(* CODESYS project tc3_physics.library
   TcLibraryId: Beckhoff Automation GmbH|Tc3_Physics|3.1.10.3
   Company: Beckhoff Automation GmbH
   DefaultNamespace: Tc3_Physics
   Version: 3.1.10.3
   Placeholder: Tc3_Physics
   Title: Tc3_Physics

Project tree, tasks and I/O mapping:
  Version/
    global variables Global_Version
  POUs/
    _Internal/
      function block IPlcGeometry2D [ST]: FB_init, FB_exit
      function block IPlcDynamicConstraint [ST]: FB_init, FB_exit
    Spatial/
      Positions/
        function block PositionXY [ST]: FB_init, FB_reinit, FB_exit, SetZero, SetValues, SetValuesXY, SetValuesRP, GetRadius, GetPhi, Invert, ConcatenateWith, ShiftByXY, x, y
        function block PositionXYC [ST]: FB_init, FB_reinit, FB_exit, SetZero, SetValues, SetValuesXY, SetValuesXYC, Invert, ConcatenateWith, StepByLocalXY, ShiftByXY, TurnByC, Transform, x, y, c
    Dynamics/
      function block DynamicConstraint_Container [ST]: FB_init, FB_exit, Clear, AddConstraint, Count
      function block DynamicConstraint_PathXY [ST]: FB_init, FB_exit, SetValuesVADJ, V, A, D, J
      function block DynamicConstraint_Path [ST]: FB_init, FB_exit
      function block DynamicConstraint_Coordinates [ST]: FB_init, FB_exit, AddLimit, SetLimit, RemoveLimit, Clear, GetV, GetA, GetD, GetJ, Count
    Coordinates/
      function GetMcsCoordinateType [ST]
  DUTs/
    Enumerations/
      data type E_RotationCoordinates
      data type E_CoordCategory
      data type E_McsCoordType
    data type CoordinateType
  GVLs/
    global variables GVL
*)

// DUTs/CoordinateType

(* Coordinate type. Use provided constants such as Coord_Mcs_X or factory functions such as GetMcsCoordinateType for creation. *)
	{attribute 'TcIecLibraryType'}
{attribute 'Namespace' := 'MC'}
TYPE CoordinateType : 
	STRUCT
		(* Reserved. *)
		{attribute 'hide'}
		_reserved0 : ULINT := 0;
	END_STRUCT
END_TYPE

// DUTs/Enumerations/E_RotationCoordinates

(* Enumeration of rotation conventions. 
          The order of letters defines the order of rotation around local axes.
          This also defines order in which user should program rotation values. *)
	{attribute 'TcIecLibraryType'}
{attribute 'qualified_only'}
{attribute 'strict'}
TYPE E_RotationCoordinates : (
	ABC:=0, 	(* ABC *)
	ACB:=1, 	(* ACB *)
	BCA:=2, 	(* BCA *)
	BAC:=3, 	(* BAC *)
	CAB:=4, 	(* CAB *)
	CBA:=5, 	(* CBA *)
	ABA:=6, 	(* ABA *)
	ACA:=7, 	(* ACA *)
	BAB:=8, 	(* BAB *)
	BCB:=9, 	(* BCB *)
	CAC:=10, 	(* CAC *)
	CBC:=11	(* CBC *)
) UDINT;
END_TYPE

// DUTs/Enumerations/E_CoordCategory

(* Enumeration coordinate categories. *)
	{attribute 'TcIecLibraryType'}
{attribute 'qualified_only'}
{attribute 'strict'}
TYPE E_CoordCategory : (
	Invalid:=16#0, 	(* Invalid *)
	MCS:=16#1, 	(* MCS *)
	ACS:=16#2, 	(* ACS *)
	Uninterpreted:=16#3	(* Uninterpreted *)
) UDINT;
END_TYPE

// DUTs/Enumerations/E_McsCoordType

(* Enumeration of MCS coordinate types. *)
	{attribute 'TcIecLibraryType'}
{attribute 'qualified_only'}
{attribute 'strict'}
TYPE E_McsCoordType : (
	Invalid:=16#0, 	(* Invalid *)
	X:=16#11, 	(* X *)
	Y:=16#21, 	(* Y *)
	Z:=16#31, 	(* Z *)
	A1:=16#41, 	(* A1 *)
	A2:=16#42, 	(* A2 *)
	A3:=16#43, 	(* A3 *)
	B1:=16#51, 	(* B1 *)
	B2:=16#52, 	(* B2 *)
	B3:=16#53, 	(* B3 *)
	C1:=16#61, 	(* C1 *)
	C2:=16#62, 	(* C2 *)
	C3:=16#63	(* C3 *)
) UDINT;
END_TYPE

// Version/Global_Version
{attribute 'TcGenerated'}
// This function has been automatically generated from the project information.
VAR_GLOBAL CONSTANT
	{attribute 'const_non_replaced'}
	{attribute 'linkalways'}
	stLibVersion_Tc3_Physics : ST_LibVersion := (iMajor := 3, iMinor := 1, iBuild := 10, iRevision := 3, sVersion := '3.1.10.3');
	{attribute 'const_non_replaced'}
	{attribute 'linkalways'}
	sLibraryId_Tc3_Physics : String := 'Beckhoff Automation GmbH|Tc3_Physics|3.1.10.3';
END_VAR

// GVLs/GVL

VAR_GLOBAL CONSTANT
		Coord_Mcs_X	:	CoordinateType := GetMcsCoordinateType(E_McsCoordType.X);
		Coord_Mcs_Y	:	CoordinateType := GetMcsCoordinateType(E_McsCoordType.Y);
		Coord_Mcs_Z	:	CoordinateType := GetMcsCoordinateType(E_McsCoordType.Z);
		Coord_Mcs_A1	:	CoordinateType := GetMcsCoordinateType(E_McsCoordType.A1);
		Coord_Mcs_A2	:	CoordinateType := GetMcsCoordinateType(E_McsCoordType.A2);
		Coord_Mcs_A3	:	CoordinateType := GetMcsCoordinateType(E_McsCoordType.A3);
		Coord_Mcs_B1	:	CoordinateType := GetMcsCoordinateType(E_McsCoordType.B1);
		Coord_Mcs_B2	:	CoordinateType := GetMcsCoordinateType(E_McsCoordType.B2);
		Coord_Mcs_B3	:	CoordinateType := GetMcsCoordinateType(E_McsCoordType.B3);
		Coord_Mcs_C1	:	CoordinateType := GetMcsCoordinateType(E_McsCoordType.C1);
		Coord_Mcs_C2	:	CoordinateType := GetMcsCoordinateType(E_McsCoordType.C2);
		Coord_Mcs_C3	:	CoordinateType := GetMcsCoordinateType(E_McsCoordType.C3);
	END_VAR

// POUs/_Internal/IPlcGeometry2D

	{attribute 'c++_compatible'}
	{attribute 'external_name' := 'IPlcGeometry2D_GUID_10E0F6A8_63F4_E8DF_FC4C_04BB1E5E2A5A'}
	{attribute 'TcIecLibraryType'}
	{attribute 'no_explicit_call' :='do not call this POU directly'}
	{attribute 'no_assign_warning'}
	(* Internal representation of an object in the planar space. *)
	FUNCTION_BLOCK IPlcGeometry2D
	VAR
		(* x-coordinate of the instance. *)
		px : LREAL;
		(* y-coordinate of the instance. *)
		py : LREAL;
		(* c-rotation of the instance given in degrees [°]. *)
		pc : LREAL;
		 {attribute 'hide'}
		_reserved1 : ARRAY [1..24] OF USINT;
	END_VAR
	VAR_OUTPUT
		(* ErrorCode for last method execution *)
		nErrorId : UDINT;
		(* Error during last method execution *)
		bError : BOOL;
	END_VAR
	VAR
		 {attribute 'hide'}
		_reserved2 : ARRAY [1..35] OF USINT;
	END_VAR


	(* Internal method *)
	{attribute 'hide'}
	METHOD FB_init : BOOL
	VAR_INPUT
		(*  if TRUE, the retain variables are initialized (warm start / cold start) *)
		bInitRetains : BOOL;
		(*  if TRUE, the instance afterwards gets moved into the copy code (online change) *)
		bInCopyCode : BOOL;
	END_VAR
END_METHOD


	(* Internal method *)
	{attribute 'hide'}
	METHOD FB_exit : BOOL
	VAR_INPUT
		(*  if TRUE, the exit method is called for exiting an instance that is copied afterwards (online change). *)
		bInCopyCode : BOOL;
	END_VAR
END_METHOD

END_FUNCTION_BLOCK

// POUs/_Internal/IPlcDynamicConstraint

	{attribute 'c++_compatible'}
	{attribute 'external_name' := 'IPlcDynamicConstraint_GUID_3FC1F02B_4572_E019_EEF1_2A289E49A8C4'}
	{attribute 'TcIecLibraryType'}
	{attribute 'no_explicit_call' := 'do not call this POU directly'}
	(* Internal representation of dynamic constraints. *)
	FUNCTION_BLOCK IPlcDynamicConstraint
	VAR
		{attribute 'hide'}
		_reserved0 : ULINT;
		 {attribute 'hide'}
		_reserved1 : UINT_0_32;
		 {attribute 'hide'}
		_reserved2 : ARRAY [1..4] OF UINT_8_16;
		 {attribute 'hide'}
		_reserved3 : ARRAY [1..20] OF USINT;
	END_VAR


	(* Internal method *)
	{attribute 'hide'}
	METHOD FB_init : BOOL
	VAR_INPUT
		(*  if TRUE, the retain variables are initialized (warm start / cold start) *)
		bInitRetains : BOOL;
		(*  if TRUE, the instance afterwards gets moved into the copy code (online change) *)
		bInCopyCode : BOOL;
	END_VAR
END_METHOD


	(* Internal method *)
	{attribute 'hide'}
	METHOD FB_exit : BOOL
	VAR_INPUT
		(*  if TRUE, the exit method is called for exiting an instance that is copied afterwards (online change). *)
		bInCopyCode : BOOL;
	END_VAR
END_METHOD

END_FUNCTION_BLOCK

// POUs/Dynamics/DynamicConstraint_Container

	{attribute 'c++_compatible'}
	{attribute 'external_name' := 'DynamicConstraint_Container_GUID_5BE2A102_DEC2_E8C2_FA36_46962A4D76F7'}
	{attribute 'TcIecLibraryType'}
	{attribute 'no_explicit_call' := 'do not call this POU directly'}
	(* A container for dynamic constraints. *)
	FUNCTION_BLOCK DynamicConstraint_Container EXTENDS IPlcDynamicConstraint


	(* Internal method *)
	{attribute 'hide'}
	METHOD FB_init : BOOL
	VAR_INPUT
		(*  if TRUE, the retain variables are initialized (warm start / cold start) *)
		bInitRetains : BOOL;
		(*  if TRUE, the instance afterwards gets moved into the copy code (online change) *)
		bInCopyCode : BOOL;
	END_VAR
END_METHOD


	(* Internal method *)
	{attribute 'hide'}
	METHOD FB_exit : BOOL
	VAR_INPUT
		(*  if TRUE, the exit method is called for exiting an instance that is copied afterwards (online change). *)
		bInCopyCode : BOOL;
	END_VAR
END_METHOD


	(* Removes all dynamic constraints from the container. *)
	METHOD Clear
END_METHOD


	(* Adds a dynamic constraint to the container. *)
	METHOD AddConstraint
	VAR_INPUT
		(* A reference to the constraint to be added. *)
 {attribute 'GUID' := '3FC1F02B-4572-E019-EEF1-2A289E49A8C4'}
				Constraint : REFERENCE TO IPlcDynamicConstraint;
	END_VAR
END_METHOD


{attribute 'monitoring' := 'call'}
	PROPERTY Count : UDINT
GET
END_GET
END_PROPERTY

END_FUNCTION_BLOCK

// POUs/Dynamics/DynamicConstraint_PathXY

	{attribute 'c++_compatible'}
	{attribute 'external_name' := 'DynamicConstraint_PathXY_GUID_93F1DCD9_4C66_E87D_E5F9_729BDE55A4DD'}
	{attribute 'TcIecLibraryType'}
	{attribute 'no_explicit_call' := 'do not call this POU directly'}
	(* One dimensional dynamic constraint along the XY-components of a path, ignoring non-tangential effects. *)
	FUNCTION_BLOCK DynamicConstraint_PathXY EXTENDS IPlcDynamicConstraint 
	VAR
		 {attribute 'hide'}
		_reserved1_1 : ARRAY [1..8] OF USINT;
	END_VAR


	(* Internal method *)
	{attribute 'hide'}
	METHOD FB_init : BOOL
	VAR_INPUT
		(*  if TRUE, the retain variables are initialized (warm start / cold start) *)
		bInitRetains : BOOL;
		(*  if TRUE, the instance afterwards gets moved into the copy code (online change) *)
		bInCopyCode : BOOL;
	END_VAR
END_METHOD


	(* Internal method *)
	{attribute 'hide'}
	METHOD FB_exit : BOOL
	VAR_INPUT
		(*  if TRUE, the exit method is called for exiting an instance that is copied afterwards (online change). *)
		bInCopyCode : BOOL;
	END_VAR
END_METHOD


	(* Set the dynamic limits of this instance. *)
	METHOD SetValuesVADJ
	VAR_INPUT
		(* Maximum velocity. *)
 {attribute 'GUID' := '0100FF8A-3F83-4535-990A-614CFBA4DA63'}
		 {attribute 'Namespace' := 'MC'}
				V : MC_LREAL;
		(* Maximum acceleration. *)
 {attribute 'GUID' := '0100FF8A-3F83-4535-990A-614CFBA4DA63'}
		 {attribute 'Namespace' := 'MC'}
				A : MC_LREAL;
		(* Maximum deceleration. *)
 {attribute 'GUID' := '0100FF8A-3F83-4535-990A-614CFBA4DA63'}
		 {attribute 'Namespace' := 'MC'}
				D : MC_LREAL;
		(* Maximum jerk. *)
 {attribute 'GUID' := '0100FF8A-3F83-4535-990A-614CFBA4DA63'}
		 {attribute 'Namespace' := 'MC'}
				J : MC_LREAL;
	END_VAR
END_METHOD


{attribute 'monitoring' := 'call'}
	PROPERTY V : MC_LREAL
SET
END_SET
GET
END_GET
END_PROPERTY


{attribute 'monitoring' := 'call'}
	PROPERTY A : MC_LREAL
SET
END_SET
GET
END_GET
END_PROPERTY


{attribute 'monitoring' := 'call'}
	PROPERTY D : MC_LREAL
SET
END_SET
GET
END_GET
END_PROPERTY


{attribute 'monitoring' := 'call'}
	PROPERTY J : MC_LREAL
SET
END_SET
GET
END_GET
END_PROPERTY

END_FUNCTION_BLOCK

// POUs/Dynamics/DynamicConstraint_Path

	{attribute 'c++_compatible'}
	{attribute 'external_name' := 'DynamicConstraint_Path_GUID_80B0EF21_0090_E8B9_D392_32033FD4307F'}
	{attribute 'TcIecLibraryType'}
	{attribute 'hide'}
	{attribute 'no_explicit_call' := 'do not call this POU directly'}
	(* DEPRECATED. Please replace with either DynamicConstraint_PathXY or DynamicConstraint_Coordinates, depending on use case. *)
	FUNCTION_BLOCK DynamicConstraint_Path EXTENDS DynamicConstraint_PathXY


	(* Internal method *)
	{attribute 'hide'}
	METHOD FB_init : BOOL
	VAR_INPUT
		(*  if TRUE, the retain variables are initialized (warm start / cold start) *)
		bInitRetains : BOOL;
		(*  if TRUE, the instance afterwards gets moved into the copy code (online change) *)
		bInCopyCode : BOOL;
	END_VAR
END_METHOD


	(* Internal method *)
	{attribute 'hide'}
	METHOD FB_exit : BOOL
	VAR_INPUT
		(*  if TRUE, the exit method is called for exiting an instance that is copied afterwards (online change). *)
		bInCopyCode : BOOL;
	END_VAR
END_METHOD

END_FUNCTION_BLOCK

// POUs/Dynamics/DynamicConstraint_Coordinates

	{attribute 'c++_compatible'}
	{attribute 'external_name' := 'DynamicConstraint_Coordinates_GUID_D4374861_1791_E449_FC85_9407145F2147'}
	{attribute 'TcIecLibraryType'}
	{attribute 'no_explicit_call' := 'do not call this POU directly'}
	(* Dynamic constraints for individual coordinates. *)
	FUNCTION_BLOCK DynamicConstraint_Coordinates EXTENDS IPlcDynamicConstraint


	(* Internal method *)
	{attribute 'hide'}
	METHOD FB_init : BOOL
	VAR_INPUT
		(*  if TRUE, the retain variables are initialized (warm start / cold start) *)
		bInitRetains : BOOL;
		(*  if TRUE, the instance afterwards gets moved into the copy code (online change) *)
		bInCopyCode : BOOL;
	END_VAR
END_METHOD


	(* Internal method *)
	{attribute 'hide'}
	METHOD FB_exit : BOOL
	VAR_INPUT
		(*  if TRUE, the exit method is called for exiting an instance that is copied afterwards (online change). *)
		bInCopyCode : BOOL;
	END_VAR
END_METHOD


	(* Adds limits for a specific coordinate. If the coordinate is already limited, limits are merged. *)
	METHOD AddLimit
	VAR_INPUT
		(* Coordinate type. E.g. Coord_Mcs_X, Coord_Mcs_Y, ... *)
 {attribute 'GUID' := 'ABF37E9D-1614-4226-99CD-162368D15A32'}
		 {attribute 'Namespace' := 'MC'}
				Coordinate : CoordinateType;
		(* Maximum velocity. *)
 {attribute 'GUID' := '0100FF8A-3F83-4535-990A-614CFBA4DA63'}
		 {attribute 'Namespace' := 'MC'}
				V : MC_LREAL;
		(* Maximum acceleration. *)
 {attribute 'GUID' := '0100FF8A-3F83-4535-990A-614CFBA4DA63'}
		 {attribute 'Namespace' := 'MC'}
				A : MC_LREAL;
		(* Maximum deceleration. *)
 {attribute 'GUID' := '0100FF8A-3F83-4535-990A-614CFBA4DA63'}
		 {attribute 'Namespace' := 'MC'}
				D : MC_LREAL;
		(* Maximum jerk. *)
 {attribute 'GUID' := '0100FF8A-3F83-4535-990A-614CFBA4DA63'}
		 {attribute 'Namespace' := 'MC'}
				J : MC_LREAL;
	END_VAR
END_METHOD


	(* Sets limits for a specific coordinate. If the coordinate is already limited, existing limits are overwritten. *)
	METHOD SetLimit
	VAR_INPUT
		(* Coordinate type. E.g. Coord_Mcs_X, Coord_Mcs_Y, ... *)
 {attribute 'GUID' := 'ABF37E9D-1614-4226-99CD-162368D15A32'}
		 {attribute 'Namespace' := 'MC'}
				Coordinate : CoordinateType;
		(* Maximum velocity. *)
 {attribute 'GUID' := '0100FF8A-3F83-4535-990A-614CFBA4DA63'}
		 {attribute 'Namespace' := 'MC'}
				V : MC_LREAL;
		(* Maximum acceleration. *)
 {attribute 'GUID' := '0100FF8A-3F83-4535-990A-614CFBA4DA63'}
		 {attribute 'Namespace' := 'MC'}
				A : MC_LREAL;
		(* Maximum deceleration. *)
 {attribute 'GUID' := '0100FF8A-3F83-4535-990A-614CFBA4DA63'}
		 {attribute 'Namespace' := 'MC'}
				D : MC_LREAL;
		(* Maximum jerk. *)
 {attribute 'GUID' := '0100FF8A-3F83-4535-990A-614CFBA4DA63'}
		 {attribute 'Namespace' := 'MC'}
				J : MC_LREAL;
	END_VAR
END_METHOD


	(* Removes limits for a specific coordinate. *)
	METHOD RemoveLimit
	VAR_INPUT
		(* Coordinate type. E.g. Coord_Mcs_X, Coord_Mcs_Y, ... *)
 {attribute 'GUID' := 'ABF37E9D-1614-4226-99CD-162368D15A32'}
		 {attribute 'Namespace' := 'MC'}
				Coordinate : CoordinateType;
	END_VAR
END_METHOD


	(* Removes limits for all coordinates. *)
	METHOD Clear
END_METHOD


	(* Gets the contained velocity limit for a specific coordinate. If no limits for the coordinate are set, returns MC_INVALID. *)
	METHOD GetV : MC_LREAL
	VAR_INPUT
		(* Coordinate type. E.g. Coord_Mcs_X, Coord_Mcs_Y, ... *)
 {attribute 'GUID' := 'ABF37E9D-1614-4226-99CD-162368D15A32'}
		 {attribute 'Namespace' := 'MC'}
				Coordinate : CoordinateType;
	END_VAR
END_METHOD


	(* Gets the contained acceleration limit for a specific coordinate. If no limits for the coordinate are set, returns MC_INVALID. *)
	METHOD GetA : MC_LREAL
	VAR_INPUT
		(* Coordinate type. E.g. Coord_Mcs_X, Coord_Mcs_Y, ... *)
 {attribute 'GUID' := 'ABF37E9D-1614-4226-99CD-162368D15A32'}
		 {attribute 'Namespace' := 'MC'}
				Coordinate : CoordinateType;
	END_VAR
END_METHOD


	(* Gets the contained deceleration limit for a specific coordinate. If no limits for the coordinate are set, returns MC_INVALID. *)
	METHOD GetD : MC_LREAL
	VAR_INPUT
		(* Coordinate type. E.g. Coord_Mcs_X, Coord_Mcs_Y, ... *)
 {attribute 'GUID' := 'ABF37E9D-1614-4226-99CD-162368D15A32'}
		 {attribute 'Namespace' := 'MC'}
				Coordinate : CoordinateType;
	END_VAR
END_METHOD


	(* Gets the contained jerk limit for a specific coordinate. If no limits for the coordinate are set, returns MC_INVALID. *)
	METHOD GetJ : MC_LREAL
	VAR_INPUT
		(* Coordinate type. E.g. Coord_Mcs_X, Coord_Mcs_Y, ... *)
 {attribute 'GUID' := 'ABF37E9D-1614-4226-99CD-162368D15A32'}
		 {attribute 'Namespace' := 'MC'}
				Coordinate : CoordinateType;
	END_VAR
END_METHOD


{attribute 'monitoring' := 'call'}
	PROPERTY Count : UDINT
GET
END_GET
END_PROPERTY

END_FUNCTION_BLOCK

// POUs/Coordinates/GetMcsCoordinateType

	{attribute 'TcIecLibraryType'}
	{attribute 'external_name' := 'GetMcsCoordinateType_GUID_655639B8_F48A_EF5D_FEC5_B9E3E765F48B'}
	(* Creates a CoordinateType FB from E_McsCoordType. *)
	FUNCTION GetMcsCoordinateType : CoordinateType
	VAR_INPUT
		mcsType	:	E_McsCoordType;	(* Mcs coordinate type. *)
	END_VAR

END_FUNCTION

// POUs/Spatial/Positions/PositionXY

	{attribute 'c++_compatible'}
	{attribute 'external_name' := 'PositionXY_GUID_C46347E0_12C2_E7BB_C81D_74646ABD268D'}
	{attribute 'TcIecLibraryType'}
	{attribute 'no_explicit_call' :='do not call this POU directly'}
	{attribute 'no_assign_warning'}
	(* Position in the 2D Cartesian space. *)
	FUNCTION_BLOCK PositionXY EXTENDS IPlcGeometry2D


	(* Internal method *)
	{attribute 'hide'}
	METHOD FB_init : BOOL
	VAR_INPUT
		(*  if TRUE, the retain variables are initialized (warm start / cold start) *)
		bInitRetains : BOOL;
		(*  if TRUE, the instance afterwards gets moved into the copy code (online change) *)
		bInCopyCode : BOOL;
	END_VAR
END_METHOD


	(* Internal method *)
	{attribute 'hide'}
	METHOD FB_reinit : BOOL
END_METHOD


	(* Internal method *)
	{attribute 'hide'}
	METHOD FB_exit : BOOL
	VAR_INPUT
		(*  if TRUE, the exit method is called for exiting an instance that is copied afterwards (online change). *)
		bInCopyCode : BOOL;
	END_VAR
END_METHOD


	(* Set the coordinates of this position to '0.0'. *)
	METHOD SetZero
END_METHOD


	(* Set the coordinates of this position. *)
	METHOD SetValues
	VAR_IN_OUT
		(* The coordinate values to set. *)
 {attribute 'GUID' := 'C46347E0-12C2-E7BB-C81D-74646ABD268D'}
				positionXY : PositionXY;
	END_VAR
END_METHOD


	(* Set the xy-coordinates of this position. *)
	METHOD SetValuesXY
	VAR_INPUT
		(* x-component of the position. *)
		x : LREAL;
		(* y-component of the position. *)
		y : LREAL;
	END_VAR
END_METHOD


	(* Set the components of this position in polar coordinates. *)
	METHOD SetValuesRP
	VAR_INPUT
		(* Distance from the origin. *)
		radius : LREAL;
		(* Polar angle of this position in degrees [°]. *)
		phi : LREAL;
	END_VAR
END_METHOD


	(* Get the distance from the origin. *)
	METHOD GetRadius : LREAL
END_METHOD


	(* Get the polar angle scaled in degrees [°]. *)
	METHOD GetPhi : LREAL
END_METHOD


	(* Invert this position. *)
	METHOD Invert
END_METHOD


	(* Concatenate with a 2nd position. *)
	METHOD ConcatenateWith
	VAR_IN_OUT
		(* The 2nd position to concatenate with. *)
 {attribute 'GUID' := 'C46347E0-12C2-E7BB-C81D-74646ABD268D'}
				position : PositionXY;
	END_VAR
END_METHOD


	(* Displace the components of this position. *)
	METHOD ShiftByXY
	VAR_INPUT
		(* Shift of the x-component of this position. *)
		dx : LREAL;
		(* Shift of the y-component of this position. *)
		dy : LREAL;
	END_VAR
END_METHOD


	PROPERTY x : LREAL
SET
END_SET
GET
END_GET
END_PROPERTY


	PROPERTY y : LREAL
SET
END_SET
GET
END_GET
END_PROPERTY

END_FUNCTION_BLOCK

// POUs/Spatial/Positions/PositionXYC

	{attribute 'c++_compatible'}
	{attribute 'external_name' := 'PositionXYC_GUID_4159FE5D_7F20_EFFD_DD32_3790E42CC33F'}
	{attribute 'TcIecLibraryType'}
	{attribute 'no_explicit_call' :='do not call this POU directly'}
	{attribute 'no_assign_warning'}
	(* A position in the xy-plane with an in-plane direction c. *)
	FUNCTION_BLOCK PositionXYC EXTENDS IPlcGeometry2D


	(* Internal method *)
	{attribute 'hide'}
	METHOD FB_init : BOOL
	VAR_INPUT
		(*  if TRUE, the retain variables are initialized (warm start / cold start) *)
		bInitRetains : BOOL;
		(*  if TRUE, the instance afterwards gets moved into the copy code (online change) *)
		bInCopyCode : BOOL;
	END_VAR
END_METHOD


	(* Internal method *)
	{attribute 'hide'}
	METHOD FB_reinit : BOOL
END_METHOD


	(* Internal method *)
	{attribute 'hide'}
	METHOD FB_exit : BOOL
	VAR_INPUT
		(*  if TRUE, the exit method is called for exiting an instance that is copied afterwards (online change). *)
		bInCopyCode : BOOL;
	END_VAR
END_METHOD


	(* Set the components of this vector to '0.0'. *)
	METHOD SetZero
END_METHOD


	(* Set the components of this position. *)
	METHOD SetValues
	VAR_IN_OUT
		(* The values to set. *)
 {attribute 'GUID' := '4159FE5D-7F20-EFFD-DD32-3790E42CC33F'}
				positionXYC : PositionXYC;
	END_VAR
END_METHOD


	(* Set the spatial components of this position. *)
	METHOD SetValuesXY
	VAR_INPUT
		(* x-component of the position. *)
		x : LREAL;
		(* y-component of the position. *)
		y : LREAL;
	END_VAR
END_METHOD


	(* Set the components of this position. *)
	METHOD SetValuesXYC
	VAR_INPUT
		(* x-component of the position. *)
		x : LREAL;
		(* y-component of the position. *)
		y : LREAL;
		(* c-component of the position scaled in degrees [°]. *)
		c : LREAL;
	END_VAR
END_METHOD


	(* Invert this position. *)
	METHOD Invert
END_METHOD


	(* Multiply this position by a 2nd from the right. *)
	METHOD ConcatenateWith
	VAR_IN_OUT
		(* The position to concatenate with. *)
 {attribute 'GUID' := '4159FE5D-7F20-EFFD-DD32-3790E42CC33F'}
				position : PositionXYC;
	END_VAR
END_METHOD


	(* Apply a local step in respect to the local coordinate frame without changing the orientation. *)
	METHOD StepByLocalXY
	VAR_INPUT
		(* The displacement within the local x-direction. *)
		dx : LREAL;
		(* The displacement within the local y-direction. *)
		dy : LREAL;
	END_VAR
END_METHOD


	(* Displace the components of this position. *)
	METHOD ShiftByXY
	VAR_INPUT
		(* Shift of the x-component of this position. *)
		dx : LREAL;
		(* Shift of the y-component of this position. *)
		dy : LREAL;
	END_VAR
END_METHOD


	(* Rotate the attached orientation without changing the Cartesian coodinates. *)
	METHOD TurnByC
	VAR_INPUT
		(* Angular displacement given in degrees [°]. *)
		dc : LREAL;
	END_VAR
END_METHOD


	(* Place a PositionXY into the coordinate system referenced by this position. *)
	METHOD Transform
	VAR_IN_OUT
		(* Position to transform. *)
 {attribute 'GUID' := 'C46347E0-12C2-E7BB-C81D-74646ABD268D'}
				positionXY : PositionXY;
	END_VAR
END_METHOD


	PROPERTY x : LREAL
SET
END_SET
GET
END_GET
END_PROPERTY


	PROPERTY y : LREAL
SET
END_SET
GET
END_GET
END_PROPERTY


	PROPERTY c : LREAL
SET
END_SET
GET
END_GET
END_PROPERTY

END_FUNCTION_BLOCK
